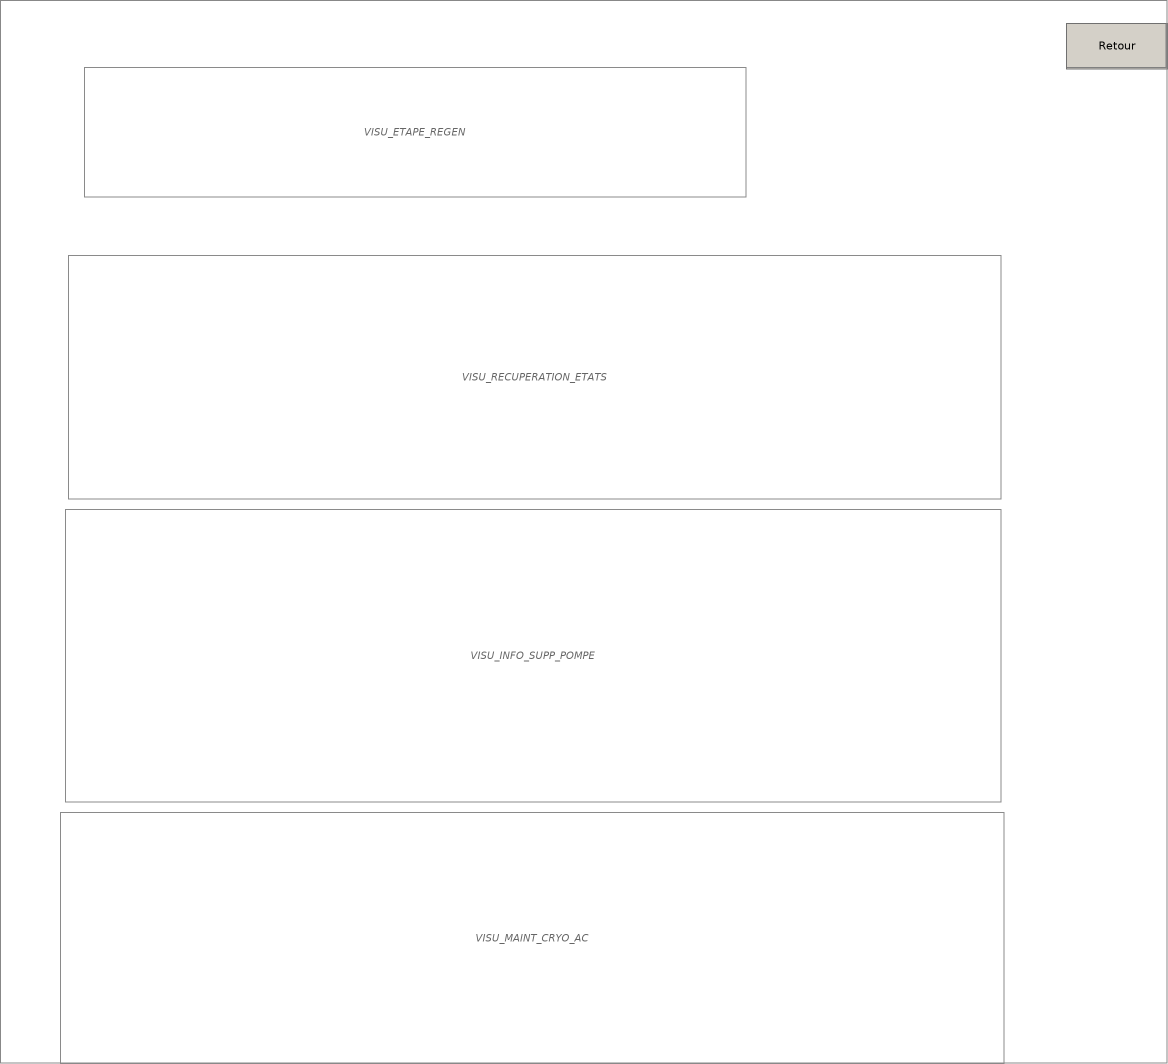
VISUALIZATION VISU_INFO  // 1168x1064
VAR_IN_OUT
	m_Input_CRYO: BLOCK_RS232_ONBOARD_V4;
	m_Input_PRG_POMPAGE: BLOCK_PRG_POMPAGE;
END_VAR
    Button (1066,23 102x46), "Retour", text list: 'GlabalTextList', text index: 16
        OnMouseClick: change screen: Previous SYN_POMPAGE
        OnMouseClick: execute { .VISU_INDEX_MANU := 0; }
    Frame (60,812 944x252), invisible if: NOT Global_Variables.PRG_USER.MANUFACTURER, input disabled if: NOT Global_Variables.PRG_USER.ACTU_USER.CONF_MACHINE OR NOT Global_Variables.PRG_USER.MANUFACTURER
        shows VISU_MAINT_CRYO_AC(COM := m_Input_CRYO)
    Frame (65,509 936x293)
        shows VISU_INFO_SUPP_POMPE(COM := m_Input_CRYO)
    Frame (68,255 933x244)
        shows VISU_RECUPERATION_ETATS(COM := m_Input_CRYO)
    Frame (84,67 662x130)
        shows VISU_ETAPE_REGEN(COM := m_Input_CRYO)
END_VISUALIZATION

(* stored: Version 1.1.0.1, ProductVersion 3.1.4026.18
   Visu VISU_INFO: Id {a63b1ed8-752d-4b74-a532-2a25d8e06cf0} *)
